TEXTLIST TextList
  0 = 'Option1'
  1 = 'Option2'
  2 = 'Option3'
  3 = 'Option4'
  4 = 'Option5'
   = ''
END_TEXTLIST

(* stored: Version 1.1.0.1, ProductVersion 3.1.4024.4
   TextList TextList: Id {68ea4962-3db0-474c-9df0-163cdcf682e9} *)
